# EPICS substitutions: epics/m-epics-eemcu/eemcuApp/Db/TwoAxis-m2.substitutions
file "eemcu.template"
{
pattern
{P,       N,  M,   R,      DTYP,         PORT,     ADDR,  DESC,       EGU, DIR,  VELO, JVEL,  JAR,  VBAS,  ACCL,  BDST, DLY,  BVEL,  BACC,  MRES,      ERES,       PREC,  DLLM,  DHLM,  INIT}
{"IOC:",  2,  m2, m2-,    "asynMotor",   MCU1,     2,   "motor 2",    mm,  Pos,  24.9, 10,    10.2, 0,     1,     0,    0.3,  1,     .2,   0.0046875, 0.01754386,  3,   12000, 120000,    ""}
}
